// TIA Portal project "Machine Tool Coolant Control" (V17)
// Machine Tool Coolant Control
// The coolant should activate when the machine tool starts and continue for 5 sec after the tool stops. The Machine tool will operate for 10 sec with a break of 5 sec.

(* hardware
DEVICE "S7-1200 station_1"  S7-1200 Station
   slot 0: "Rack_0"  S7-1200 Rack  Rack  V1.0
   slot 1: "PLC_1"  CPU 1215C AC/DC/Rly  6ES7 215-1BG40-0XB0  V4.5
*)

// ===== PLC "PLC_1"  CPU 1215C AC/DC/Rly =====

VAR_GLOBAL   // PLC tag table "Default tag table"
   "Machine_Bench_Turn_ON_Switch" AT %I0.0 : Bool;
   "Coolant" AT %Q0.0 : Bool;
   "Machine" AT %Q0.1 : Bool;
   "Tag_1" AT %M0.2 : Bool;
   "Tag_2" AT %M0.0 : Bool;
   "Tag_3" AT %M0.1 : Bool;
END_VAR

// folder: System blocks/Program resources

DATA_BLOCK "IEC_Timer_0_DB"   // DB1
{ S7_Optimized_Access := 'TRUE' }
AUTHOR : Simatic
FAMILY : IEC
NAME : IEC_TMR
VERSION : 1.0
// stored: InstanceOfName IEC_TIMER
"IEC_TIMER"
BEGIN
END_DATA_BLOCK

DATA_BLOCK "IEC_Timer_0_DB_1"   // DB2
{ S7_Optimized_Access := 'TRUE' }
AUTHOR : Simatic
FAMILY : IEC
NAME : IEC_TMR
VERSION : 1.0
// stored: InstanceOfName IEC_TIMER
"IEC_TIMER"
BEGIN
END_DATA_BLOCK

DATA_BLOCK "IEC_Timer_0_DB_2"   // DB3
{ S7_Optimized_Access := 'TRUE' }
AUTHOR : Simatic
FAMILY : IEC
NAME : IEC_TMR
VERSION : 1.0
// stored: InstanceOfName IEC_TIMER
"IEC_TIMER"
BEGIN
END_DATA_BLOCK

DATA_BLOCK "IEC_Timer_0_DB_3"   // DB4
{ S7_Optimized_Access := 'TRUE' }
AUTHOR : Simatic
FAMILY : IEC
NAME : IEC_TMR
VERSION : 1.0
// stored: InstanceOfName IEC_TIMER
"IEC_TIMER"
BEGIN
END_DATA_BLOCK

// folder: (top level)

ORGANIZATION_BLOCK "Main"   // OB1, LAD, ProgramCycle
TITLE = "Main Program Sweep (Cycle)"
{ S7_Optimized_Access := 'TRUE' }
VERSION : 0.1
   VAR_INPUT
      Initial_Call : Bool;   // Initial call of this OB
      Remanence : Bool;   // =True, if remanent data are available
   END_VAR
BEGIN

REGION Network 1
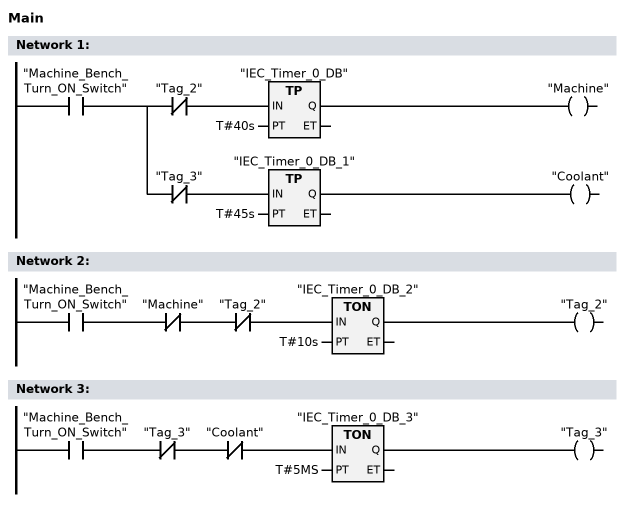
   "IEC_Timer_0_DB".TP(IN := "Machine_Bench_Turn_ON_Switch" AND NOT "Tag_2", PT := T#40s);
   "Machine" := "IEC_Timer_0_DB".Q;
   "IEC_Timer_0_DB_1".TP(IN := "Machine_Bench_Turn_ON_Switch" AND NOT "Tag_3", PT := T#45s);
   "Coolant" := "IEC_Timer_0_DB_1".Q;
END_REGION

REGION Network 2
   "IEC_Timer_0_DB_2".TON(IN := "Machine_Bench_Turn_ON_Switch" AND NOT "Machine" AND NOT "Tag_2", PT := T#10s);
   "Tag_2" := "IEC_Timer_0_DB_2".Q;
END_REGION

REGION Network 3
   "IEC_Timer_0_DB_3".TON(IN := "Machine_Bench_Turn_ON_Switch" AND NOT "Tag_3" AND NOT "Coolant", PT := T#5MS);
   "Tag_3" := "IEC_Timer_0_DB_3".Q;
END_REGION
END_ORGANIZATION_BLOCK